TYPE HMI_MAN_TemplateMachinePart :
STRUCT
	;
END_STRUCT
END_TYPE

(* stored: Version 1.1.0.1
   DUT HMI_MAN_TemplateMachinePart: Id {811c2c62-376c-4b21-b642-8a80912fe820} *)
